// TIA Portal V16 export
// export: Created 2021-09-01T13:50:45.7188082Z, ExportSetting WithDefaults, DisplayName Totally Integrated Automation Portal, DisplayVersion V16 Update 3, DisplayName TIA Portal Version Control Interface, DisplayVersion V16 Update 2, DisplayName TIA Portal Openness, DisplayVersion V16 Update 3, DisplayName TIA Portal Teamcenter Gateway, DisplayVersion V16, DisplayName STEP 7 Professional, DisplayVersion V16 Update 3, DisplayName STEP 7 Safety, DisplayVersion V16, DisplayName WinCC Advanced, DisplayVersion V16 Update 3
TYPE "DevInStack"
// stored: IsFailsafeCompliant false
   STRUCT
      Dev : Int;   // Номер машины
      TimeDev : Time;   // Время наработки
   END_STRUCT;
END_TYPE
